TYPE ST_AxisControl :
STRUCT
    //Actions from controls system
    bExecute: BOOL; //Rising edge to execute some motion FB's
    bReset: BOOL; //Reset axis from Error state
    bStop: BOOL;
    bEnable: BOOL; //Enable axis drive
    bJogFwd: BOOL;
    bJogBwd: BOOL;
	eCommand: E_MotionFunctions;
END_STRUCT
END_TYPE

(* stored: Version 1.1.0.1, ProductVersion 3.1.4024.0
   DUT ST_AxisControl: Id {c02b2c99-be98-4acd-b0cb-dc10c1ff77f2} *)
